# B&R Automation Studio project SemProj-F26-PLC
Automation Studio 4.9

## Configuration Config1

### Task classes (Cpu.sw)
```
Cyclic#1 (cycle 1000 us, tolerance 1000 us):
  Prog_1ms <- Prog_1ms.prg
Cyclic#2 (cycle 10000 us, tolerance 10000 us):
  Obs_10ms <- Obs_10ms.prg
Binaries: udbdef, FWRules, TCData, sysconf, Role, User, iomap, ashwd, asfw, arconfig, ashwac
Libraries: standard, runtime, astime, asieccon
```

### Hardware
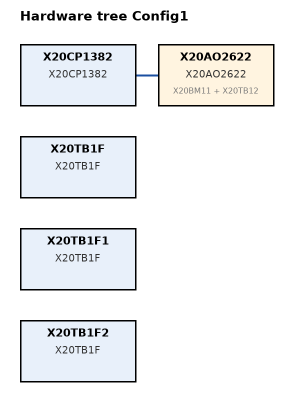
```
X20AO2622 : X20AO2622 v1.3.0.0  [SS1 -> X20TB12.SS; SL -> X20BM11.SL1]
X20BM11 : X20BM11 v1.1.0.0  [X2X1 -> X20CP1382.IF6]
X20CP1382 : X20CP1382 v1.15.0.0  [X1 -> X1.SL; X2 -> X2.SL; X3 -> X3.SL]
  Module X1 (Type=X1, Virtual=true, Version=1.15.0.0)
    Connection (Connector=SS1, TargetModule=X20TB1F, TargetConnector=SS)
    Connection (Connector=SL, TargetModule=X20CP1382, TargetConnector=X1)
  Module X2 (Type=X2, Virtual=true, Version=1.15.0.0)
    Connection (Connector=SS1, TargetModule=X20TB1F1, TargetConnector=SS)
    Connection (Connector=SL, TargetModule=X20CP1382, TargetConnector=X2)
    X2CounterFunction = AB
    X2CounterTimeInfo = 32Bit
  Module X3 (Type=X3, Virtual=true, Version=1.15.0.0)
    Connection (Connector=SS1, TargetModule=X20TB1F2, TargetConnector=SS)
    Connection (Connector=SL, TargetModule=X20CP1382, TargetConnector=X3)
  Connector IF2:
    ActivateDevice = 1
    Mode = Manual
    InternetAddress = 192.168.8.101
    SubnetMask = 255.255.255.0
    InaNodeNumber = 0
  Connector IF3:
    CycleTime = 1000
  ConfigurationID = spro4_pendulum_Config1
  SystemTick = 1000
  TaskClassIdleTime = 1000
  Cyclic1Duration = 1000
  Cyclic1Tolerance = 1000
  Cyclic2Duration = 10000
  Cyclic2Tolerance = 10000
X20TB12 : X20TB12 v1.0.0.0
X20TB1F : X20TB1F v1.0.0.0
X20TB1F1 : X20TB1F v1.0.0.0
X20TB1F2 : X20TB1F v1.0.0.0
```

## Logical view

Binary libraries used (declarations not repeated): operator, runtime, astime, AsIecCon, standard, AsOpcUas, AsOpcUac

### Global.var - Global variables
```iecst
VAR
	I_pos_pendulum_rad : REAL;
	SI_estop_B : BOOL;
	SI_estop_A : BOOL;
	SI_reset_btn : BOOL;
	I_drive_active : BOOL;
	I_drive_no_fault : BOOL;
	I_endstop_negative : BOOL;
	I_endstop_positive : BOOL;
	I_pos_cart : DINT;
	I_pos_pendulum : DINT;
	Q_drive_enable : BOOL;
	Q_drive_faultreset : BOOL;
	Q_drive_operating_mode : BOOL;
	Q_vel_cart : INT;
	Q_reset_LED : BOOL;
	reset_cart_position : BOOL;
	reset_pendulum_position : BOOL;
	A : ARRAY[0..3,0..3] OF REAL := [1.0,0.009535,0.0000575,0.0000002737,0.0,0.9085,-0.01132,0.00003438,0.0,0.001945,1.002,0.009989,0.0,0.3829,0.4582,0.9986];
	B : ARRAY[0..3] OF REAL := [0.001859,0.366,-0.007782,-1.531];
	K : ARRAY[0..3] OF REAL := [-9.97788845498053,-4.33797239803683,-8.31962221505295,-1.27391028745717];
	u : REAL;
	xGlobal : ARRAY[0..3] OF REAL;
	x_out : ARRAY[0..3] OF REAL;
	theta_smoothed : REAL;
	x_smoothed : REAL;
	theta_last : REAL;
	u_smoothed : REAL;
	u_last : REAL;
	Pi : REAL := 3.1415926535;
	length : DINT;
	xGlobalAvged : ARRAY[0..3] OF REAL;
	x : ARRAY[0..3] OF REAL;
END_VAR
```


### Program Logical/Prog_10ms (IEC)

#### Variables.var
```iecst
VAR
	temp_pendulum_pos : DINT;
	Temp_checker : REAL;
	length : DINT;
	led_ton : TON;
	cart_velocity : INT;
	length_calibration_steps : USINT;
	d1 : REAL;
	calibration_finished : BOOL;
	centering_in_progress : BOOL;
	pos_pendulum_absolute : DINT;
	d2 : REAL;
	pos_pendulum_deg : REAL;
	pos_pendulum_rad : REAL;
	pendulum_position_rad_last : REAL;
	K_In : ARRAY[0..2] OF REAL := [-9.32952485563385,-53.0199254837238,-0.386299598154963];
	K_Out : ARRAY[0..2] OF REAL := [0.033376485856261,0.00205473985473051,0.131363047248811];
	pendulum_velocity_rad : REAL;
	cart_position_last : REAL;
	pend_vel_b : REAL;
	pend_vel_a : REAL;
	i : INT;
	j : INT;
	stop_acc : DINT;
	cart_velocity_calculated : REAL;
	pos_cart_mm : DINT;
	target_position : DINT;
	new_cart_velocity : INT;
	stopped : BOOL;
	balancing_active : BOOL;
	length_mm : DINT;
	swingup_complete : BOOL;
	Swing_movement : Position_case;
	pos_cart : DINT;
	eOut : ARRAY[0..2] OF REAL;
	eIn : ARRAY[0..2] OF REAL;
	uIn : ARRAY[0..2] OF REAL;
	springforce : REAL;
	controllerType : USINT;
	uSmoothingConst : REAL;
	xSmoothingConst : REAL;
	thetaSmoothingConst : REAL;
	uOut : ARRAY[0..2] OF REAL;
	tempTimer : DINT;
END_VAR
```

#### Main.st
```iecst
PROGRAM _INIT
	cart_velocity := 5000;
	Q_vel_cart := 0;
	length := 0;
	Q_drive_enable  := FALSE;
	length_calibration_steps := 5;
	calibration_finished := FALSE;
	centering_in_progress := FALSE;
	Temp_checker := 0;
	stop_acc := 400;
	stopped := FALSE;
	balancing_active := FALSE;
	Swing_movement := position0;
	thetaSmoothingConst := 0.25;
	xSmoothingConst := 0.25;
	uSmoothingConst := 0.25;
	i := 0;
	controllerType := 2;
	springforce := 0.5;
	tempTimer := 0;

	FOR i := 0 TO 2 DO
		eOut[i] := 0;
		eIn[i] := 0;
		uOut[i] := 0;
		uIn[i] := 0;
	END_FOR

END_PROGRAM

PROGRAM _CYCLIC

	// Handle EStop
	IF(SI_estop_A AND SI_estop_B) THEN
		Q_drive_enable := TRUE;
	ELSE
		Q_drive_enable  := FALSE;
		Q_reset_LED := FALSE;
	END_IF

	// Handle Reset Btn
	IF(SI_reset_btn) THEN
		Q_drive_faultreset := NOT Q_drive_faultreset;
	ELSIF I_drive_no_fault THEN
		Q_reset_LED := TRUE;
	ELSE
		led_ton(IN:=NOT led_ton.Q, PT := T#200ms);
		IF(led_ton.Q) THEN
			Q_reset_LED := NOT Q_reset_LED;
			Q_reset_LED := NOT Q_reset_LED;
		END_IF
	END_IF

	pos_cart := I_pos_cart;
	I_pos_pendulum_rad := ((I_pos_pendulum - 2048) / 4096.0) * 2 * Pi;
	pos_pendulum_absolute := I_pos_pendulum MOD 4096;
	IF(pos_pendulum_absolute < 0) THEN
		pos_pendulum_absolute := pos_pendulum_absolute + 4096;
	END_IF
	pos_pendulum_deg := (pos_pendulum_absolute - 2048) / 4096.0 * 360.0;
	pos_pendulum_rad := (pos_pendulum_absolute - 2048) / 4096.0 * 2 * Pi;
	pos_cart_mm := pos_cart / 240;
	length_mm := length / 240;
	cart_velocity_calculated := (pos_cart_mm - cart_position_last) / 0.01;
	pendulum_velocity_rad := (I_pos_pendulum_rad - pendulum_position_rad_last) / 0.01;

	x[0] := - pos_cart_mm / 1000.0 + length_mm / 2000.0;
	x[1] := - cart_velocity_calculated / 1000.0;
	x[2] := pos_pendulum_rad;
	x[3] := pendulum_velocity_rad;

	IF(length_calibration_steps = 5) THEN
		reset_pendulum_position := TRUE;
		length_calibration_steps := 4;
		reset_cart_position := TRUE;
		reset_cart_position := FALSE;
	ELSIF(length_calibration_steps = 4) THEN
		reset_pendulum_position := FALSE;
		Q_vel_cart := -cart_velocity;
		Q_drive_faultreset := NOT Q_drive_faultreset;
		IF (NOT I_endstop_negative) THEN
			Q_vel_cart := 0;
			reset_cart_position := TRUE;

			tempTimer := tempTimer + 1;

			IF(tempTimer > 500) THEN
				length_calibration_steps := 3;
			END_IF
		END_IF
	ELSIF(length_calibration_steps = 3) THEN
		reset_cart_position := FALSE;
		Q_vel_cart := cart_velocity;
		Q_drive_faultreset := NOT Q_drive_faultreset;
		length_calibration_steps := 2;
	ELSIF(length_calibration_steps = 2) THEN
		Q_drive_faultreset := NOT Q_drive_faultreset;
		IF (NOT I_endstop_positive) THEN
			Q_vel_cart := 0;
			length := MAX(length, pos_cart);
			length_calibration_steps := 1;
		END_IF
	ELSIF(length_calibration_steps = 1) THEN
		Q_vel_cart := -cart_velocity;
		Q_drive_faultreset := NOT Q_drive_faultreset;
		length_calibration_steps := 0;
	END_IF

	IF(NOT swingup_complete AND length_calibration_steps = 0) THEN
		target_position :=  length / 2;
		IF(ABS(pos_cart - target_position) < stop_acc) THEN
			Q_vel_cart := 0;
			swingup_complete := TRUE;
		ELSIF(pos_cart < target_position) THEN
			Q_vel_cart := REAL_TO_INT(cart_velocity * 1.0);
			Q_drive_faultreset := NOT Q_drive_faultreset;
		ELSIF(pos_cart > target_position) THEN
			Q_vel_cart := REAL_TO_INT(-cart_velocity * 1.0);
			Q_drive_faultreset := NOT Q_drive_faultreset;
		END_IF
	END_IF

	IF(swingup_complete AND NOT stopped) THEN

		eOut[2] := eOut[1];
		eOut[1] := eOut[0];
		eIn[2] := eIn[1];
		eIn[1] := eIn[0];
		uOut[2] := uOut[1];
		uOut[1] := uOut[0];
		uIn[2] := uIn[1];
		uIn[1] := uIn[0];

		(*
		eOut[0] := - x[0];
		uOut[0] := 1.924 * uOut[1] - 0.9235 * uOut[2] + 1.038 * eOut[0] - 2.073 * eOut[1] + 1.035 * eOut[2];

		IF(uOut[0] > 0.2) THEN
			uOut[0] := 0.2;
		END_IF
		IF(uOut[0] < - 0.2) THEN
			uOut[0] := - 0.2;
		END_IF

		theta_smoothed := thetaSmoothingConst * theta_smoothed + (1 - thetaSmoothingConst) * x[2];

		eIn[0] := uOut[0] - x[2];
		uIn[0] := 0.0515 * uIn[1] + 0.9485 * uIn[2] - 84.6 * eIn[0] + 150.9 * eIn[1] - 66.51 * eIn[2];*)

		eOut[0] :=  x[0];
		d1 := (eOut[0] - eOut[1]) / 0.01;
		uOut[0] := K_Out[0] * eOut[0] + K_Out[1] * (eOut[0] * 0.01) + K_Out[2] * d1;
		//uOut[0] := LIMIT(-0.2, uOut[0], 0.2);

		//eIn[0] := uOut[0] - x[2];
		eIn[0] := -x[2];
		d2 := (eIn[0] - eIn[1]) / 0.01;
		uIn[0] := K_In[0] * eIn[0] + K_In[1] * (eIn[0] * 0.01) + K_In[2] * d2;
		//uIn[0] := LIMIT(-1, uIn[0], 1);

		IF(controllerType = 1) THEN
			u := 0;
			FOR i:= 0 TO 3 BY 1 DO
				u := u - K[i] * x[i];
			END_FOR
		ELSE
			u := uIn[0];
		END_IF

		IF(ABS(u) < 1) THEN
			balancing_active := TRUE;
		ELSIF(ABS(u) >= 10) THEN
			Temp_checker := Temp_checker + 1;
			balancing_active := FALSE;
			(* FOR i := 0 TO 2 DO
				eOut[i] := 0;
				eIn[i] := 0;
				uOut[i] := 0;
				uIn[i] := 0;
			END_FOR *)
		END_IF

		IF(balancing_active) THEN
			new_cart_velocity := REAL_TO_INT( - 2000 * u - 2000 * (springforce * x[0]));
			IF(ABS(new_cart_velocity) < 20000) THEN
				Q_vel_cart := new_cart_velocity;
			ELSE
				IF(new_cart_velocity < 0) THEN
					Q_vel_cart := -20000;
				ELSE
					Q_vel_cart := 20000;
				END_IF
			END_IF
		ELSE
			Q_vel_cart := 0;
		END_IF

		IF(pos_cart_mm < 50 OR length_mm - pos_cart_mm < 50) THEN
			stopped := TRUE;
			Q_vel_cart := 0;
		END_IF
		IF(NOT I_endstop_positive OR NOT I_endstop_negative) THEN
			stopped := TRUE;
			Q_vel_cart := 0;
		END_IF

	END_IF

	u_last := u;
	theta_last := x[2];
	cart_position_last := pos_cart_mm;
	pendulum_position_rad_last := I_pos_pendulum_rad;

END_PROGRAM

PROGRAM _EXIT
	(* Insert code here *)

END_PROGRAM
```

### Program Logical/Prog_1ms (IEC)

#### Types.typ
```iecst
TYPE
	Swingup_State :
		(
		Swingup_Center,
		Accelerate,
		Swingup_Complete,
		Start_Swingup
		);
	Pendulum_State :
		(
		Stopped,
		Balancing,
		Reset,
		Swingup,
		Calibrating
		);
	Calibration_State :
		(
		Calibration_Complete,
		Calibration_Center,
		Move_Right,
		Reset_Position,
		Move_Left,
		Start_Calibration
		);
	Balancing_State :
		(
		Classic1ms,
		Classic10ms,
		Cascade1ms,
		Cascade10ms,
		PolePlacement1ms,
		PolePlacement10ms
		);
END_TYPE
```

#### Variables.var
```iecst
VAR
	SystemState : Pendulum_State;
	CalibrationState : Calibration_State;
	SwingupState : Swingup_State;
	BalancingState : Balancing_State;
	systemStateFailure : BOOL := FALSE;
	calibrationStateFailure : BOOL := FALSE;
	swingupStateFailure : BOOL := FALSE;
	balancingStateFailure : BOOL := FALSE;
	i : INT;
	j : INT;
	cartVelocity : INT := 5000;
	lengthLocal : DINT;
	stopAcc : INT := 400;
	led_ton : TON;
	lengthMm : DINT;
	cartPos : DINT;
	cartPosMm : DINT;
	cartVelCalculated : REAL;
	pendulumPosAbsolute : DINT;
	pendulumPosRad : REAL;
	pendulumVel : REAL;
	pendulumVelRad : REAL;
	data : ARRAY[0..3] OF REAL;
	cartPosLast : DINT;
	pendulumPosLast : ARRAY[0..9] OF DINT;
	errorString : STRING[80];
	iterationCounter : DINT;
	swingupPolarity : SINT;
	swingupVel : INT;
	pendulumPolarity : SINT;
	dataBacklog : ARRAY[0..9,0..3] OF REAL;
	data10ms : ARRAY[0..3] OF REAL;
	balancingActive : BOOL;
	newCartVelocity : INT;
	viableBacklog : INT;
END_VAR
```

#### Main.st
```iecst
PROGRAM _INIT
	Q_vel_cart := 0;
	SystemState := Calibrating;
	CalibrationState := Start_Calibration;
	SwingupState := Start_Swingup;
	BalancingState := Classic10ms;
	iterationCounter := 0;
	i := 1;

	(*
	xSmoothingConst := 0.25;
	uSmoothingConst := 0.25;
	thetaSmoothingConst := 0.25;
	controllerType := 2;
	springforce := 0.5;
	*)
END_PROGRAM

PROGRAM _CYCLIC

	IF(SI_estop_A AND SI_estop_B) THEN
		Q_drive_enable := TRUE;
	ELSE
		Q_drive_enable  := FALSE;
		Q_reset_LED := FALSE;
	END_IF

	IF(SI_reset_btn) THEN
		Q_drive_faultreset := NOT Q_drive_faultreset;
	ELSIF I_drive_no_fault THEN
		Q_reset_LED := TRUE;
	ELSE
		led_ton(IN:=NOT led_ton.Q, PT := T#200ms);
		IF(led_ton.Q) THEN
			Q_reset_LED := NOT Q_reset_LED;
			Q_reset_LED := NOT Q_reset_LED;
		END_IF
	END_IF

	iterationCounter := iterationCounter + 1;
	lengthMm := length / 240;
	cartPos := I_pos_cart;
	cartPosMm := cartPos / 240;
	cartVelCalculated := (cartPos - cartPosLast) * 1000.0 / 240;
	pendulumPosAbsolute := I_pos_pendulum MOD 4096;
	IF(pendulumPosAbsolute < 0) THEN
		pendulumPosAbsolute := pendulumPosAbsolute + 4096;
	END_IF
	pendulumPosRad := (pendulumPosAbsolute - 2048) / 4096.0 * 2 * Pi;
	pendulumVel := (I_pos_pendulum - pendulumPosLast[9]) / 4096.0 * 1000.0 / 10;
	pendulumVelRad := pendulumVel * 2 * Pi;

	data[0] := (cartPosMm - lengthMm / 2) / 1000.0;
	data[1] := cartVelCalculated / 1000.0;
	data[2] := pendulumPosRad;
	data[3] := pendulumVelRad;
	FOR i := 0 TO 3 DO
		xGlobal[i] := data[i];
	END_FOR

	IF(SystemState <> Calibrating) THEN
		IF(data[3] > 15 OR cartPosMm < 100 OR lengthMm - cartPosMm < 100) THEN
			Q_vel_cart := 0;
			SystemState := Reset;
		ELSIF(NOT I_endstop_negative OR NOT I_endstop_positive) THEN
			Q_vel_cart := 0;
			SystemState := Stopped;
		END_IF
	END_IF

	CASE SystemState OF
		Calibrating:

			IF(iterationCounter MOD 2 = 0 AND iterationCounter > 5000) THEN

				CASE CalibrationState OF
					Start_Calibration:
						reset_pendulum_position := TRUE;
						CalibrationState := Move_Left;

					Move_Left:
						reset_pendulum_position := FALSE;
						Q_vel_cart := -cartVelocity;
						Q_drive_faultreset := NOT Q_drive_faultreset;
						IF (NOT I_endstop_negative) THEN
							Q_vel_cart := 0;
							reset_cart_position := TRUE;
							CalibrationState := Reset_Position;
						END_IF

					Reset_Position:
						reset_cart_position := FALSE;
						Q_vel_cart := cartVelocity;
						Q_drive_faultreset := NOT Q_drive_faultreset;
						CalibrationState := Move_Right;

					Move_Right:
						Q_drive_faultreset := NOT Q_drive_faultreset;
						IF (NOT I_endstop_positive) THEN
							Q_vel_cart := 0;
							length := ABS(cartPos);
							CalibrationState := Calibration_Center;
						END_IF

					Calibration_Center:
						Q_vel_cart := -cartVelocity;
						Q_drive_faultreset := NOT Q_drive_faultreset;
						IF(ABS(cartPos - length / 2) < stopAcc) THEN
							Q_vel_cart := 0;
							CalibrationState := Calibration_Complete;
						ELSE
							Q_vel_cart := REAL_TO_INT( - data[0] / ABS(data[0]) * cartVelocity);
						END_IF

					Calibration_Complete:
						SystemState := Swingup;

					ELSE
						calibrationStateFailure := TRUE;

				END_CASE
			END_IF

		Swingup:
			CASE SwingupState OF
				Swingup_Center:
					IF(ABS(cartPos - length / 2) < stopAcc) THEN
						Q_vel_cart := 0;
						SwingupState := Start_Swingup;
					ELSE
						Q_vel_cart := REAL_TO_INT( - data[0] / ABS(data[0]) * cartVelocity);
					END_IF

				Start_Swingup:
					Q_vel_cart := 5000;
					IF(ABS(data[0]) > 0.2) THEN
						SwingupState := Accelerate;
					END_IF

				Accelerate:
					IF(data[2] > Pi / 2 AND data[3] > 0 AND data[0] < 0.2) THEN
						Q_vel_cart := 5000;
					ELSIF(data[2] < - Pi / 2 AND data[3] < 0 AND data[0] > - 0.2) THEN
						Q_vel_cart := - 5000;
					ELSE
						Q_vel_cart := 0;
					END_IF

					IF(ABS(data[2]) < 0.2) THEN
						Q_vel_cart := 0;
						SwingupState := Swingup_Complete;
						SystemState := Balancing;
					END_IF

				Swingup_Complete:
					SystemState := Balancing;

				ELSE
					swingupStateFailure := TRUE;

			END_CASE

		Balancing:
			FOR i := 0 TO 8 DO
				FOR j := 0 TO 3 DO
					dataBacklog[9 - i, j] := dataBacklog[8 - i, j];
				END_FOR
			END_FOR
			FOR j := 0 TO 3 DO
				dataBacklog[0, j] := data[j];
			END_FOR

			viableBacklog := 0;
			FOR i := 1 TO 9 DO
				IF(dataBacklog[0, 2] * dataBacklog[i, 2] > 0) THEN
					viableBacklog := i;
				ELSE
					i := 9;
				END_IF
			END_FOR

			FOR i := 0 TO 3 DO
				data10ms[i] := 0;
				FOR j := 0 TO viableBacklog DO
					data10ms[i] := data10ms[i] + dataBacklog[j, i];
				END_FOR
				data10ms[i] := data10ms[i] / 10;
			END_FOR

			FOR i := 0 TO 3 DO
				xGlobalAvged[i] := data10ms[i];
			END_FOR

			u := 0;
			FOR i:= 0 TO 1 DO
				u := u + K[i] * data[i];
			END_FOR
			FOR i:= 2 TO 3 DO
				u := u - K[i] * data[i];
			END_FOR

			IF(iterationCounter MOD 10 = 0) THEN
				IF(ABS(u) < 1) THEN
					balancingActive := TRUE;
				ELSIF(ABS(u) >= 10) THEN
					balancingActive := FALSE;
				END_IF

				IF(balancingActive) THEN
					newCartVelocity := REAL_TO_INT( - 10000 * u);
					IF(ABS(newCartVelocity) < 20000) THEN
						Q_vel_cart := newCartVelocity;
					ELSE
						IF(newCartVelocity < 0) THEN
							Q_vel_cart := -20000;
						ELSE
							Q_vel_cart := 20000;
						END_IF
					END_IF
				ELSE
					Q_vel_cart := 0;
				END_IF
			END_IF

			systemStateFailure := TRUE;

		Reset:
			systemStateFailure := TRUE;

		Stopped:
			systemStateFailure := TRUE;

		ELSE
			systemStateFailure := TRUE;

	END_CASE

	cartPosLast := cartPos;
	FOR i := 0 TO 8 DO
		pendulumPosLast[9 - i] := pendulumPosLast[8 - i];
	END_FOR
	pendulumPosLast[0] := I_pos_pendulum;

END_PROGRAM

PROGRAM _EXIT
	(* Insert code here *)

END_PROGRAM
```

### Program Logical/Obs_10ms (IEC)

#### Variables.var
```iecst
VAR
	xGlobalAvgedDiff : ARRAY[0..3] OF REAL;
	xGlobalDiff : ARRAY[0..3] OF REAL;
	xLocal : ARRAY[0..3] OF REAL;
	uLocal : REAL;
	cart_velocity_calculated : REAL;
	pos_cart_mm : DINT;
	pendulum_velocity_rad : REAL;
	pos_pendulum_rad : REAL;
	stopped : BOOL;
	xSmoothingConst : REAL;
	thetaSmoothingConst : REAL;
	uSmoothingConst : REAL;
	pos_pendulum_absolute : DINT;
	pos_cart : DINT;
	i : INT;
	pos_pendulum_deg : REAL;
	balancing_active : BOOL;
	uLocalLast : REAL;
	thetaLocalLast : REAL;
	cart_position_last : REAL;
	pendulum_position_rad_last : REAL;
	length_mm : DINT;
	eOut : ARRAY[0..2] OF REAL;
	eIn : ARRAY[0..2] OF REAL;
	uIn : ARRAY[0..2] OF REAL;
	uOut : ARRAY[0..2] OF REAL;
	K_In : ARRAY[0..2] OF REAL := [-9.32952485563385,-53.0199254837238,-0.386299598154963];
	K_Out : ARRAY[0..2] OF REAL := [0.033376485856261,0.00205473985473051,0.131363047248811];
	d1 : REAL;
	d2 : REAL;
END_VAR
```

#### Main.st
```iecst
PROGRAM _INIT
	thetaSmoothingConst := 0.25;
	xSmoothingConst := 0.25;
	uSmoothingConst := 0.25;
	i := 0;

	(*FOR i := 0 TO 2 DO
		eOut[i] := 0;
		eIn[i] := 0;
		uOut[i] := 0;
		uIn[i] := 0;
	END_FOR*)

END_PROGRAM

PROGRAM _CYCLIC
	pos_cart := I_pos_cart;
	I_pos_pendulum_rad := ((I_pos_pendulum - 2048) / 4096.0) * 2 * Pi;
	pos_pendulum_absolute := I_pos_pendulum MOD 4096;
	IF(pos_pendulum_absolute < 0) THEN
		pos_pendulum_absolute := pos_pendulum_absolute + 4096;
	END_IF
	pos_pendulum_deg := (pos_pendulum_absolute - 2048) / 4096.0 * 360.0;
	pos_pendulum_rad := (pos_pendulum_absolute - 2048) / 4096.0 * 2 * Pi;
	pos_cart_mm := pos_cart / 240;
	length_mm := length / 240;
	cart_velocity_calculated := (pos_cart_mm - cart_position_last) / 0.01;
	pendulum_velocity_rad := (I_pos_pendulum_rad - pendulum_position_rad_last) / 0.01;

	xLocal[0] := - pos_cart_mm / 1000.0 + length_mm / 2000.0;
	xLocal[1] := - cart_velocity_calculated / 1000.0;
	xLocal[2] := pos_pendulum_rad;
	xLocal[3] := pendulum_velocity_rad;

	IF(NOT stopped) THEN
		eOut[2] := eOut[1];
		eOut[1] := eOut[0];
		eIn[2] := eIn[1];
		eIn[1] := eIn[0];
		uOut[2] := uOut[1];
		uOut[1] := uOut[0];
		uIn[2] := uIn[1];
		uIn[1] := uIn[0];

		(*
		eOut[0] := - x[0];
		uOut[0] := 1.924 * uOut[1] - 0.9235 * uOut[2] + 1.038 * eOut[0] - 2.073 * eOut[1] + 1.035 * eOut[2];

		IF(uOut[0] > 0.2) THEN
			uOut[0] := 0.2;
		END_IF
		IF(uOut[0] < - 0.2) THEN
			uOut[0] := - 0.2;
		END_IF

		theta_smoothed := thetaSmoothingConst * theta_smoothed + (1 - thetaSmoothingConst) * x[2];

		eIn[0] := uOut[0] - x[2];
		uIn[0] := 0.0515 * uIn[1] + 0.9485 * uIn[2] - 84.6 * eIn[0] + 150.9 * eIn[1] - 66.51 * eIn[2];*)

		eOut[0] :=  x[0];
		d1 := (eOut[0] - eOut[1]) / 0.01;
		uOut[0] := K_Out[0] * eOut[0] + K_Out[1] * (eOut[0] * 0.01) + K_Out[2] * d1;
		//uOut[0] := LIMIT(-0.2, uOut[0], 0.2);

		//eIn[0] := uOut[0] - x[2];
		eIn[0] := -x[2];
		d2 := (eIn[0] - eIn[1]) / 0.01;
		uIn[0] := K_In[0] * eIn[0] + K_In[1] * (eIn[0] * 0.01) + K_In[2] * d2;
		//uIn[0] := LIMIT(-1, uIn[0], 1);

		uLocal := 0;
		FOR i:= 0 TO 3 BY 1 DO
			uLocal := uLocal - K[i] * x[i];
		END_FOR

		IF(ABS(u) < 1) THEN
			balancing_active := TRUE;
		ELSIF(ABS(u) >= 10) THEN
			balancing_active := FALSE;
			(* FOR i := 0 TO 2 DO
				eOut[i] := 0;
				eIn[i] := 0;
				uOut[i] := 0;
				uIn[i] := 0;
			END_FOR *)
		END_IF

		(*IF(balancing_active) THEN
			new_cart_velocity := REAL_TO_INT( - 2000 * u - 2000 * (springforce * x[0]));
			IF(ABS(new_cart_velocity) < 20000) THEN
				Q_vel_cart := new_cart_velocity;
			ELSE
				IF(new_cart_velocity < 0) THEN
					Q_vel_cart := -20000;
				ELSE
					Q_vel_cart := 20000;
				END_IF
			END_IF
		ELSE
			Q_vel_cart := 0;
		END_IF*)

		(*IF(pos_cart_mm < 50 OR length_mm - pos_cart_mm < 50) THEN
			stopped := TRUE;
			Q_vel_cart := 0;
		END_IF
		IF(NOT I_endstop_positive OR NOT I_endstop_negative) THEN
			stopped := TRUE;
			Q_vel_cart := 0;
		END_IF*)

	END_IF

	FOR i := 0 TO 3 DO
		xGlobalDiff[i] := xGlobal[i] - xLocal[i];
		xGlobalAvgedDiff[i] := xGlobalAvged[i] - xLocal[i];
		IF(xGlobalDiff[i] < 0.01) THEN
			xGlobalDiff[i] := 0;
		END_IF
		IF(xGlobalAvgedDiff[i] < 0.01) THEN
			xGlobalAvgedDiff[i] := 0;
		END_IF
	END_FOR

	uLocalLast := uLocal;
	thetaLocalLast := xLocal[2];
	cart_position_last := pos_cart_mm;
	pendulum_position_rad_last := I_pos_pendulum_rad;

END_PROGRAM

PROGRAM _EXIT

END_PROGRAM
```

### Program Logical/Program

#### Variables.var
```iecst
VAR CONSTANT
	Pi : REAL := 3.1415926535;
END_VAR
VAR
	temp_pendulum_pos : DINT;
	Temp_checker : REAL;
	length : DINT;
	led_ton : TON;
	cart_velocity : INT;
	SI_reset_last : BOOL;
	allow_Q_drive_enable : BOOL;
	length_calibration_steps : USINT;
	d1_filter : ARRAY[0..2] OF REAL;
	d2_filter : ARRAY[0..2] OF REAL;
	d1 : REAL;
	O_D : REAL;
	I_D : REAL;
	counter1 : REAL;
	counter : REAL;
	P_P : REAL;
	P_I : ARRAY[0..2] OF REAL;
	P_D : REAL;
	I_P : REAL;
	uP : ARRAY[0..2] OF REAL;
	I_N : REAL := 194.847386319238;
	O_N : REAL := 7.64741103823823;
	I_I : ARRAY[0..2] OF REAL;
	O_I : ARRAY[0..2] OF REAL;
	O_P : REAL;
	calibration_finished : BOOL;
	centering_in_progress : BOOL;
	pos_pendulum_absolute : DINT;
	d2 : REAL;
	pos_pendulum_deg : REAL;
	pos_pendulum_rad : REAL;
	pendulum_position_rad_last : REAL;
	K_In : ARRAY[0..2] OF REAL := [-9.32952485563385,-53.0199254837238,-0.386299598154963];
	K_P : ARRAY[0..2] OF REAL := [-21.8208797167883, -159.979890000381, -0.598721790617152];
	K_Out : ARRAY[0..2] OF REAL := [0.033376485856261,0.00205473985473051,0.131363047248811];
	pendulum_velocity_rad : REAL;
	cart_position_last : REAL;
	pend_vel_b : REAL;
	pend_vel_a : REAL;
	i : INT;
	j : INT;
	stop_acc : DINT;
	cart_velocity_calculated : REAL;
	pos_cart_mm : DINT;
	target_position : DINT;
	new_cart_velocity : INT;
	stopped : BOOL;
	balancing_active : BOOL;
	length_mm : DINT;
	swingup_complete : BOOL;
	Swing_movement : Position_case;
	pos_cart : DINT;
	eOut : ARRAY[0..2] OF REAL;
	eIn : ARRAY[0..2] OF REAL;
	uIn : ARRAY[0..2] OF REAL;
	springforce : REAL;
	controllerType : USINT;
	uSmoothingConst : REAL;
	xSmoothingConst : REAL;
	thetaSmoothingConst : REAL;
	uOut : ARRAY[0..2] OF REAL;
END_VAR
```

#### Main.st
```iecst
PROGRAM _INIT
	(* Insert code here *)
	cart_velocity := 5000;
	Q_vel_cart := 0;
	length := 0;
	SI_reset_last := SI_reset_btn;
	allow_Q_drive_enable := FALSE;
	Q_drive_enable  := FALSE;
	length_calibration_steps := 5;
	calibration_finished := FALSE;
	centering_in_progress := FALSE;
	Temp_checker := 0;
	stop_acc := 400;
	stopped := FALSE;
	balancing_active := FALSE;
	Swing_movement := position0;
	thetaSmoothingConst := 0.25;
	xSmoothingConst := 0.25;
	uSmoothingConst := 0.25;
	i := 1;
	controllerType := 0;
	springforce := 0.5;

	FOR i := 0 TO 2 DO
		eOut[i] := 0;
		eIn[i] := 0;
		uOut[i] := 0;
		uIn[i] := 0;
	END_FOR

END_PROGRAM

PROGRAM _CYCLIC

	// Handle EStop
	IF(SI_estop_A AND SI_estop_B) THEN
		Q_drive_enable := TRUE;
	ELSE
		Q_drive_enable  := FALSE;
		Q_reset_LED := FALSE;
	END_IF

	// Handle Reset Btn
	IF(SI_reset_btn) THEN
		Q_drive_faultreset := NOT Q_drive_faultreset;
		IF(NOT SI_reset_last) THEN
			allow_Q_drive_enable := NOT allow_Q_drive_enable;
		END_IF
	ELSIF I_drive_no_fault THEN
		Q_reset_LED := TRUE;
	ELSE
		led_ton(IN:=NOT led_ton.Q, PT := T#200ms);
		IF(led_ton.Q) THEN
			Q_reset_LED := NOT Q_reset_LED;
			Q_reset_LED := NOT Q_reset_LED;
		END_IF
	END_IF

	pos_cart := -I_pos_cart;
	I_pos_pendulum_rad := ((I_pos_pendulum - 2048) / 4096.0) * 2 * Pi;
	pos_pendulum_absolute := I_pos_pendulum MOD 4096;
	IF(pos_pendulum_absolute < 0) THEN
		pos_pendulum_absolute := pos_pendulum_absolute + 4096;
	END_IF
	pos_pendulum_deg := (pos_pendulum_absolute - 2048) / 4096.0 * 360.0;
	pos_pendulum_rad := (pos_pendulum_absolute - 2048) / 4096.0 * 2 * Pi;
	pos_cart_mm := pos_cart / 264;
	length_mm := length / 264;
	cart_velocity_calculated := (pos_cart_mm - cart_position_last) / 0.01;
	pendulum_velocity_rad := (I_pos_pendulum_rad - pendulum_position_rad_last) / 0.01;

	x[0] := - pos_cart_mm / 1000.0 + length_mm / 2000.0;
	x[1] := - cart_velocity_calculated / 1000.0;
	x[2] := pos_pendulum_rad;
	x[3] := pendulum_velocity_rad;

	IF(length_calibration_steps = 5) THEN
		reset_pendulum_position := TRUE;
		length_calibration_steps := 4;
		reset_cart_position := TRUE;
		reset_cart_position := FALSE;
	ELSIF(length_calibration_steps = 4) THEN
		reset_pendulum_position := FALSE;
		Q_vel_cart := -cart_velocity;
		Q_drive_faultreset := NOT Q_drive_faultreset;
		IF (NOT I_endstop_negative) THEN
			Q_vel_cart := 0;
			reset_cart_position := TRUE;
			length_calibration_steps := 3;
		END_IF
	ELSIF(length_calibration_steps = 3) THEN
		reset_cart_position := FALSE;
		Q_vel_cart := cart_velocity;
		Q_drive_faultreset := NOT Q_drive_faultreset;
		length_calibration_steps := 2;
	ELSIF(length_calibration_steps = 2) THEN
		Q_drive_faultreset := NOT Q_drive_faultreset;
		IF (NOT I_endstop_positive) THEN
			Q_vel_cart := 0;
			length := MAX(length, pos_cart);
			length_calibration_steps := 1;
		END_IF
	ELSIF(length_calibration_steps = 1) THEN
		Q_vel_cart := -cart_velocity;
		Q_drive_faultreset := NOT Q_drive_faultreset;
		length_calibration_steps := 0;
	END_IF

	IF(NOT swingup_complete AND length_calibration_steps = 0) THEN
		target_position :=  length / 2;
		IF(ABS(pos_cart - target_position) < stop_acc) THEN
			Q_vel_cart := 0;
			swingup_complete := TRUE;
		ELSIF(pos_cart < target_position) THEN
			Q_vel_cart := REAL_TO_INT(cart_velocity * 1.0);
			Q_drive_faultreset := NOT Q_drive_faultreset;
		ELSIF(pos_cart > target_position) THEN
			Q_vel_cart := REAL_TO_INT(-cart_velocity * 1.0);
			Q_drive_faultreset := NOT Q_drive_faultreset;
		END_IF
	END_IF

	IF(swingup_complete AND NOT stopped) THEN

		eOut[2] := eOut[1];
		eOut[1] := eOut[0];
		eIn[2] := eIn[1];
		eIn[1] := eIn[0];
		uOut[2] := uOut[1];
		uOut[1] := uOut[0];
		uIn[2] := uIn[1];
		uIn[1] := uIn[0];

		O_I[1] := O_I[0];
		d1_filter[1] := d1_filter[0];
		I_I[1] := I_I[0];
		d2_filter[1] := d2_filter[0];

		(*
		eOut[0] := - x[0];
		uOut[0] := 1.924 * uOut[1] - 0.9235 * uOut[2] + 1.038 * eOut[0] - 2.073 * eOut[1] + 1.035 * eOut[2];

		IF(uOut[0] > 0.2) THEN
			uOut[0] := 0.2;
		END_IF
		IF(uOut[0] < - 0.2) THEN
			uOut[0] := - 0.2;
		END_IF

		theta_smoothed := thetaSmoothingConst * theta_smoothed + (1 - thetaSmoothingConst) * x[2];

		eIn[0] := uOut[0] - x[2];
		uIn[0] := 0.0515 * uIn[1] + 0.9485 * uIn[2] - 84.6 * eIn[0] + 150.9 * eIn[1] - 66.51 * eIn[2];*)
		eOut[0] :=  -x[0];
		O_P := K_Out[0] * eOut[0];
		O_I[0] := O_I[1] + (K_Out[1] * (eOut[0] * 0.01));
		O_I[0] := LIMIT(-0.2, O_I[0], 0.2);
		d1 := (eOut[0] - eOut[1]) / 0.01;
		//d1_filter[0] := d1_filter[1] + (0.01*O_N* (d1 - d1_filter[1]));
		O_D := K_Out[2] * d1;

		uOut[0] :=  O_P + O_I[0] + O_D;
		uOut[0] := LIMIT(-0.2, uOut[0], 0.2);

		//eIn[0] := uOut[0] - x[2];
		eIn[0] := -x[2];
		I_P := K_In[0] * eIn[0];
		I_I[0] := I_I[1] + (K_In[1] * (eIn[0] * 0.01));
		//I_I[0] :=(K_In[1] * (eIn[0] * 0.01));
		//I_I[0] := LIMIT(-0.2, I_I[0], 0.2);
		d2 := (eIn[0] - eIn[1]) / 0.01;
		//d2_filter[0] := d2_filter[1] + (0.01*I_N* (d2 - d2_filter[1]));
		I_D := K_In[2] * d2;

		uIn[0] :=  I_P + I_I[0] + I_D;
	//	eIn[0] := -x[2];
	//	d2 := (eIn[0] - eIn[1]) / 0.01;
	//	uIn[0] := K_In[0] * eIn[0] + K_In[1] * (eIn[0] * 0.01) + K_In[2] * d2;
		//uIn[0] := LIMIT(-1, uIn[0], 1);

		uP[2] := uP[1];
		uP[1] := uP[0];
		P_I[1] := P_I[0];

		P_P := K_P[0] * eIn[0];
		P_I[0] := P_I[1] + (K_P[1] * eIn[0] * 0.01);
		P_I[0] := LIMIT(-0.2, P_I[0], 0.2);
		P_P := K_P[2]*((eIn[0] - eIn[1]) / 0.01);

		uP[0] :=  P_P + P_I[0] + P_D;

		IF(controllerType = 1) THEN
			u := 0;
			FOR i:= 0 TO 3 BY 1 DO
				u := u - K[i] * x[i];
			END_FOR
		ELSIF(controllerType = 2) THEN
			u := uP[0];
		ELSE
			u := uIn[0];
		END_IF

		IF(ABS(x[2]) < 0.4) THEN
			balancing_active := TRUE;
		ELSIF(ABS(x[2]) >= 0.6) THEN
			Temp_checker := Temp_checker + 1;
			balancing_active := FALSE;
			 FOR i := 0 TO 2 DO
				eOut[i] := 0;
				eIn[i] := 0;
				uOut[i] := 0;
				uIn[i] := 0;
				I_D := 0;
				I_P := 0;
				I_I[0] := 0;
				O_D := 0;
				O_P := 0;
				O_I[0] := 0;
				d1_filter[i] := 0;
				d2_filter[i] := 0;
				d1 := 0;
				d2 := 0;
				P_P := 0;
				P_I[i] := 0;
				P_D := 0;

			END_FOR
		END_IF
		//- 2000 * (springforce * x[0])vs
		counter := 10000*x[0];
		IF(balancing_active) THEN
			new_cart_velocity := REAL_TO_INT( -10000 * u);
		(*	IF(u < 0) THEN
				counter := counter +1;
			ELSIF(u > 0) THEN
				counter1 := counter1 +1;
			END_IF*)
			IF(ABS(new_cart_velocity) < 20000) THEN
				Q_vel_cart := new_cart_velocity;
			ELSE
				IF(new_cart_velocity < 0) THEN
					Q_vel_cart := -20000;
				ELSE
					Q_vel_cart := 20000;
				END_IF
			END_IF
		ELSE
			Q_vel_cart := 0;
		END_IF

		IF(pos_cart_mm < 50 OR length_mm - pos_cart_mm < 50) THEN
			stopped := TRUE;
			Q_vel_cart := 0;
		END_IF
		IF(NOT I_endstop_positive OR NOT I_endstop_negative) THEN
			stopped := TRUE;
			Q_vel_cart := 0;
		END_IF

	END_IF

	u_last := u;
	theta_last := x[2];
	SI_reset_last := SI_reset_btn;
	cart_position_last := pos_cart_mm;
	pendulum_position_rad_last := I_pos_pendulum_rad;

END_PROGRAM

PROGRAM _EXIT
	(* Insert code here *)

END_PROGRAM
```

Listed in the project but not available here: Logical/Global.typ
